FUNCTION_BLOCK fb_RobotStatusToBools
VAR_INPUT
	statusstring : STRING;
END_VAR
VAR_OUTPUT
	baTemp : ARRAY[0..20] OF BOOL;
END_VAR
VAR
	byTemp : BYTE;
	iTemp : INT := 0;
END_VAR

FOR iTemp := 0 TO LEN(statusstring) BY 1 DO
	IF statusstring[iTemp] = 16#30 THEN
		baTemp[iTemp] := FALSE;
	ELSE
		baTemp[iTemp] := TRUE;
	END_IF
END_FOR

END_FUNCTION_BLOCK

(* stored: Version 1.1.0.1, ProductVersion 3.1.4020.3
   POU fb_RobotStatusToBools: Id {cd065c85-7eb4-4e77-839f-3233ef6844ad}, SpecialFunc None *)
